(* IEC 61131-3 sources: plc_generation_empirical_study/datasets/task_bank_v0_2/tasks/C05_B16_composite, 2 files *)

(* ---- interface.st ---- *)
FUNCTION_BLOCK C05_B16_composite
VAR_INPUT
    A_MonitorEnable : BOOL;
    A_Heartbeat : BOOL;
    A_Reset : BOOL;
    B_Start : BOOL;
    B_Stop : BOOL;
    B_Permit : BOOL;
    B_OilPressure : BOOL;
    B_MotorFeedback : BOOL;
    B_Reset : BOOL;
    SubsystemBEnable : BOOL;
    CrossReset : BOOL;
END_VAR
VAR_OUTPUT
    A_TimedOut : BOOL;
    A_Healthy : BOOL;
    B_LubePump : BOOL;
    B_MotorCommand : BOOL;
    B_Cooldown : BOOL;
    B_Fault : BOOL;
    B_State : INT;
    CrossReady : BOOL;
    CrossBlocked : BOOL;
END_VAR
END_FUNCTION_BLOCK

(* ---- reference.st ---- *)
FUNCTION_BLOCK C05_B16_composite
VAR_INPUT
    A_MonitorEnable : BOOL;
    A_Heartbeat : BOOL;
    A_Reset : BOOL;
    B_Start : BOOL;
    B_Stop : BOOL;
    B_Permit : BOOL;
    B_OilPressure : BOOL;
    B_MotorFeedback : BOOL;
    B_Reset : BOOL;
    SubsystemBEnable : BOOL;
    CrossReset : BOOL;
END_VAR
VAR_OUTPUT
    A_TimedOut : BOOL;
    A_Healthy : BOOL;
    B_LubePump : BOOL;
    B_MotorCommand : BOOL;
    B_Cooldown : BOOL;
    B_Fault : BOOL;
    B_State : INT;
    CrossReady : BOOL;
    CrossBlocked : BOOL;
END_VAR
VAR
    A_Watchdog : TON;
    B_PreLube : TON;
    B_FeedbackWait : TON;
    B_CoolTimer : TON;
END_VAR

A_Watchdog(IN := A_MonitorEnable AND (NOT A_Heartbeat) AND (NOT A_TimedOut), PT := T#400ms);
IF A_Watchdog.Q THEN
    A_TimedOut := TRUE;
ELSIF A_Reset AND (NOT A_MonitorEnable) THEN
    A_TimedOut := FALSE;
END_IF;
A_Healthy := A_MonitorEnable AND (NOT A_TimedOut);

IF CrossReset THEN
    CrossReady := FALSE;
ELSIF A_TimedOut THEN
    CrossReady := TRUE;
END_IF;
CrossBlocked := SubsystemBEnable AND (NOT CrossReady);

IF SubsystemBEnable AND CrossReady THEN
    B_PreLube(IN := (B_State = 1) AND B_OilPressure, PT := T#300ms);
    B_FeedbackWait(IN := (B_State = 2) AND (NOT B_MotorFeedback), PT := T#400ms);
    B_CoolTimer(IN := (B_State = 4), PT := T#300ms);
    IF (B_State <> 0) AND (B_State <> 4) AND (B_Stop OR (NOT B_Permit)) THEN
        B_State := 4;
    ELSIF (B_State = 3) AND (NOT B_OilPressure) THEN
        B_Fault := TRUE;
        B_State := 4;
    ELSIF (B_State = 2) AND B_FeedbackWait.Q THEN
        B_Fault := TRUE;
        B_State := 4;
    ELSIF (B_State = 0) AND B_Start AND B_Permit AND (NOT B_Stop) AND (NOT B_Fault) THEN
        B_State := 1;
    ELSIF (B_State = 1) AND B_PreLube.Q THEN
        B_State := 2;
    ELSIF (B_State = 2) AND B_MotorFeedback THEN
        B_State := 3;
    ELSIF (B_State = 4) AND B_CoolTimer.Q THEN
        B_State := 0;
    END_IF;
    IF B_Reset AND (B_State = 0) AND (NOT B_Start) THEN B_Fault := FALSE; END_IF;
    B_LubePump := ((B_State = 1) OR (B_State = 2) OR (B_State = 3) OR (B_State = 4));
    B_MotorCommand := ((B_State = 2) OR (B_State = 3)) AND (NOT B_Fault);
    B_Cooldown := (B_State = 4);
ELSE
    B_LubePump := FALSE;
    B_MotorCommand := FALSE;
    B_Cooldown := FALSE;
    B_Fault := FALSE;
    B_State := 0;
END_IF;

END_FUNCTION_BLOCK
